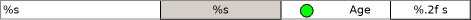
VISUALIZATION VISU_AlpacaGetBool  // 471x20
VAR_IN_OUT
	stInstance : ST_AlpacaGetBool;
END_VAR
    Rectangle (160,0 121x20), "%s", text variable: stInstance.bValue, colour toggle: stInstance.bValue
    Ellipse (300,4 13x13), colour toggle: stInstance.eStatusCode <> E_AlpacaStatusCode.OK
    Rectangle (0,0 161x20), "%s", text variable: stInstance.sName
    Rectangle (390,0 81x20), "%.2f s", text variable: stInstance.rAge
    Label (340,0 41x20), "Age"
END_VISUALIZATION

(* stored: Version 1.1.0.1, ProductVersion 3.1.4024.12
   Visu VISU_AlpacaGetBool: Id {4252a094-d74e-428a-b496-f2231ad19447} *)
